FUNCTION_BLOCK MoveRel IMPLEMENTS I_MoveRel
VAR
	mcMoveRel : MC_MoveRelative;
END_VAR
VAR_IN_OUT
	Axis : AXIS_REF;
END_VAR

mcMoveRel(Axis := Axis);

PROPERTY Acceleration : MC_LREAL
GET
Acceleration := mcMoveRel.Acceleration;
END_GET
SET
mcMoveRel.Acceleration := Acceleration;
END_SET
END_PROPERTY

PROPERTY BufferMode : MC_Buffermode
GET
BufferMode := mcMoveRel.BufferMode;
END_GET
SET
mcMoveRel.BufferMode := BufferMode;
END_SET
END_PROPERTY

PROPERTY Busy : BOOL
GET
Busy := mcMoveRel.Busy;
END_GET
END_PROPERTY

PROPERTY Deceleration : MC_LREAL
GET
Deceleration := mcMoveRel.Deceleration;
END_GET
SET
mcMoveRel.Deceleration := Deceleration;
END_SET
END_PROPERTY

PROPERTY Distance : MC_LREAL
GET
Distance := mcMoveRel.Distance;
END_GET
SET
mcMoveRel.Distance := Distance;
END_SET
END_PROPERTY

PROPERTY Done : BOOL
GET
Done := mcMoveRel.Done;
END_GET
END_PROPERTY

PROPERTY Error : BOOL
GET
Error := mcMoveRel.Error;
END_GET
END_PROPERTY

PROPERTY Execute : BOOL
GET
Execute := mcMoveRel.Execute;
END_GET
SET
mcMoveRel.Execute := Execute;
END_SET
END_PROPERTY

PROPERTY Jerk : MC_LREAL
GET
Jerk := mcMoveRel.Jerk;
END_GET
SET
mcMoveRel.Jerk := Jerk;
END_SET
END_PROPERTY

PROPERTY Velocity : MC_LREAL
GET
Velocity := mcMoveRel.Velocity;
END_GET
SET
mcMoveRel.Velocity := Velocity;
END_SET
END_PROPERTY

END_FUNCTION_BLOCK

(* stored: Version 1.1.0.1
   POU MoveRel: Id {9ca1e6f1-5c27-40c7-9f76-999c535b3f26}, SpecialFunc None
   Property Acceleration: Id {7ecc5ab3-15ae-4024-a4ef-a8f5ac0b8b93}
   Get Get: Id {72d76dae-a4d9-43ce-b149-b49bae071284}
   Set Set: Id {278cec4c-3132-4aaa-b447-b81c4c7f10c8}
   Property BufferMode: Id {5915dfae-a5ae-4d40-b309-4b53a8d3982f}
   Get Get: Id {2f23724a-8cea-4b53-9823-3bd430970efe}
   Set Set: Id {d9f89a99-81f8-457c-8e22-facc958ceb06}
   Property Busy: Id {7c23e43e-bc2f-4735-b223-4adec3827db5}
   Get Get: Id {73cce52d-291c-4327-aa1e-2a73f5d42bf4}
   Property Deceleration: Id {4fb840b1-7736-4a60-b91a-afe7bfc85c3c}
   Get Get: Id {a206fc7d-d2d3-47a9-a20a-db58787edcad}
   Set Set: Id {e818e475-6fed-45a0-905f-23ed767cbcac}
   Property Distance: Id {be786d34-ebd2-4f73-8b06-f39f08222532}
   Get Get: Id {02cce890-a4b2-4b99-866b-a04a978b19bc}
   Set Set: Id {4ca77e39-a9fe-4fb1-b5b3-414adb6d732d}
   Property Done: Id {6c125584-0b98-4f70-9a46-06087d551624}
   Get Get: Id {7bad797f-f078-4525-a2c5-345ba5a7ed7a}
   Property Error: Id {cdfdf972-5601-440e-8469-8be8334b5d4a}
   Get Get: Id {4c5f9990-6836-4ced-8980-0bc120364fca}
   Property Execute: Id {13bbac01-af0a-4c88-9b13-5f106b671973}
   Get Get: Id {1b7cce1d-f7f7-4dca-ad61-cba6d312219c}
   Set Set: Id {267e852f-b7b1-4a72-8f58-813b8b3f7500}
   Property Jerk: Id {000417e2-abe0-48ae-8e70-6f4397424a06}
   Get Get: Id {1eac950f-6cd1-4236-b538-a6ac1547a731}
   Set Set: Id {82ca6325-50a3-43d0-a691-58593405761e}
   Property Velocity: Id {b60bb925-7261-4bcc-a818-57fca7c480c8}
   Get Get: Id {4fd17538-7f44-4607-8fff-0627ca88fc6c}
   Set Set: Id {2e3242a1-18b3-469f-b955-e9a6a6b3e657} *)
